// TIA Portal V17 export
// export: Created 2024-09-27T18:48:51.098157Z, ExportSetting WithDefaults, DisplayName Totally Integrated Automation Portal, DisplayVersion V17, DisplayName TIA Portal Openness, DisplayVersion V17, DisplayName TIA Portal Version Control Interface, DisplayVersion V17, DisplayName STEP 7 Professional, DisplayVersion V17, DisplayName STEP 7 Safety, DisplayVersion V17, DisplayName WinCC Professional, DisplayVersion V17
VAR_GLOBAL   // PLC tag table "Default tag table"
   i_PB_RESET_BEZPIECZENSTWA AT %I0.0 : Bool;
   i_KURTYNA_ŚWIETLNA_OK AT %I0.1 : Bool;
   i_E_STOP_OK AT %I0.2 : Bool;
   i_PB_START AT %I0.3 : Bool;
   i_PB_STOP AT %I0.4 : Bool;
   i_SIŁOWNIK_ZACISKAJĄCY_UGÓRY AT %I0.5 : Bool;
   i_SIŁOWNIK_ZACISKAJĄCY_W_DOLE AT %I0.6 : Bool;
   "i_SIŁOWNIK NASTAWY_GŁĘBOKIE" AT %I0.7 : Bool;
   "i_SIŁOWNIK NASTAWY _PŁYTKIE" AT %I1.0 : Bool;
   i_SIŁOWNIK_ODBIORU_POZ_STÓŁ AT %I1.1 : Bool;
   i_SIŁOWNIK_ODBIORU_POZ_ZRZUT AT %I1.2 : Bool;
   i_CZUJNIK_POZYCJI_STOŁU AT %I1.3 : Bool;
   i_CZUJNIK_SZTUKI_OK AT %I1.4 : Bool;
   i_CZUJNIK_PŁYTKIE_PRZÓD AT %I1.5 : Bool;
   Axis_1_Drive_IN AT %I68.0 : "PD_TEL3_IN";
   q_GŁÓWNY_ZAWÓR_POWIETRZA_ON AT %Q0.0 : Bool;
   q_NIEBIESKA_LAMPKA_SAFETY AT %Q0.1 : Bool;
   q_SIŁOWNIK_ZACISKAJĄCY_DOL AT %Q0.2 : Bool;
   q_EJECTOR_VACUM AT %Q0.3 : Bool;
   q_SIŁOWNIK_ZMIANY_GŁĘBOKIE AT %Q0.4 : Bool;
   q_EJECTOR_BLOWOFF AT %Q0.5 : Bool;
   q_SIŁOWNIK_ODBIERAJĄCY_STÓŁ AT %Q0.6 : Bool;
   q_LED_LAMP AT %Q0.7 : Bool;
   q_REZERWA1 AT %Q1.0 : Bool;
   q_REZERWA2 AT %Q1.1 : Bool;
   q_CZERWONA_KOLUMNA_SYGNALIZACYJNA AT %Q8.0 : Bool;
   q_ZÓŁTA_KOLUMNA_SYGNALIZACYJNA AT %Q8.1 : Bool;
   q_ZIELONA_KOLUMNA_SYGNALIZACYJNA AT %Q8.2 : Bool;
   q_BUZZER_KOLUMNA_SYGNALIZACYJNA AT %Q8.3 : Bool;
   q_SAFETY_RELAY_RESET AT %Q8.4 : Bool;
   q_REZERWA4 AT %Q8.5 : Bool;
   q_REZERWA5 AT %Q8.6 : Bool;
   q_REZERWA6 AT %Q8.7 : Bool;
   Clock_Byte AT %MB0 : Byte;
   Clock_10Hz AT %M0.0 : Bool;
   Clock_5Hz AT %M0.1 : Bool;
   "Clock_2.5Hz" AT %M0.2 : Bool;
   Clock_2Hz AT %M0.3 : Bool;
   "Clock_1.25Hz" AT %M0.4 : Bool;
   Clock_1Hz AT %M0.5 : Bool;
   "Clock_0.625Hz" AT %M0.6 : Bool;
   "Clock_0.5Hz" AT %M0.7 : Bool;
   m_SAFETY_OK AT %M1.0 : Bool;
   m_AUTO_MODE AT %M1.1 : Bool;
   m_SERVO_READY AT %M1.2 : Bool;
   MAN_SIŁ_ZAG_GÓRA AT %M1.3 : Bool;
   MAN_SIŁ_ZAG_DÓŁ AT %M1.4 : Bool;
   MAN_SIŁ_NASTAWY_GŁĘBOKIE AT %M1.5 : Bool;
   MAN_SIŁ_NASTAWY_PŁYTKIE AT %M1.6 : Bool;
   MAN_SIŁ_ODBIOR_STÓŁ AT %M1.7 : Bool;
   MAN_SIŁ_ODBIOR_ZRZUT AT %M2.0 : Bool;
   MAN_JOG_STOL_FWD AT %M2.1 : Bool;
   MAN_JOG_STOL_BWD AT %M2.2 : Bool;
   MAN_POZYCJA_STÓŁ_FWD AT %M2.3 : Bool;
   MAN_POZYCJA_STÓŁ_BWD AT %M2.4 : Bool;
   MAN_EJECTOR_SSANIE AT %M2.5 : Bool;
   MAN_EJECTOR_PRZEDMUCH AT %M2.6 : Bool;
   TP_ZAPISZ_WARTOŚĆ_PRED AT %M2.7 : Bool;
   TP_ZAPISZ_WARTOŚĆ_CZASU_PRZEDMUCHU AT %M3.0 : Bool;
   TP_ZAPISZ_WARTOSC_CZASU_SSANIA AT %M3.1 : Bool;
   TP_AKT_PRED_STOŁU AT %MW4 : Int;
   TP_NOWA_PRED_STOŁU AT %MW6 : Int;
   TP_AKT_CZAS_PRZEDMUCHU AT %MD50 : DInt;
   TP_NOWY_CZAS_PRZEDMUCHU AT %MD54 : DInt;
   TP_AKT_CZAS_SSANIA AT %MD58 : DInt;
   TP_NOWY_CZAS_SSANIA AT %MD62 : DInt;
   TP_LICZNIK_CAŁKOWITY AT %MD16 : DInt;
   TP_LICZNIK_ZADANE AT %MD20 : DInt;
   TP_LICZNIK_WYKONANE AT %MD24 : DInt;
   TP_KASUJ_LICZNIK_ZADANE AT %M3.2 : Bool;
   TP_USTAW_LICZNIK_ZADANE AT %M3.3 : Bool;
   TP_KASUJ_LICZNIK_AKTUALNE AT %M3.4 : Bool;
   m_STOL_KAT_OBROTU AT %MW28 : Int;
   TP_LED_ZAŁĄCZ AT %M3.5 : Bool;
   m_SRV_STO_ON AT %M3.6 : Bool;
   TP_USTAW_CZAS_TAKTU AT %M3.7 : Bool;
   AUTO_NUMER_KROKU AT %MW30 : Int;
   AUTO_KROK_1_ZAŁADUNEK AT %M32.0 : Bool;
   AUTO_KROK_2_OBRÓT_USTAW_GŁĘBOKIE AT %M32.1 : Bool;
   AUTO_KROK_3_ROZŁADUNEK AT %M32.2 : Bool;
   AUTO_KROK_4_ZJAZD_GŁĘBOKIE AT %M32.3 : Bool;
   AUTO_KROK_5_OBRÓT_USTAW_PLYTKIE AT %M32.4 : Bool;
   "AUTO_KROK_6_ZJAZD GŁOWICY PŁYTKIE" AT %M32.5 : Bool;
   AUTO_SERVO_FWD AT %M34.0 : Bool;
   AUTO_SIŁOWNIK_ZACISKAJĄCY_DÓŁ AT %M34.1 : Bool;
   AUTO_SIŁOWNIK_ZACISKAJĄCY_GÓRA AT %M34.2 : Bool;
   AUTO_SIŁOWNIK_NASTAWY_GŁĘBOKIE AT %M34.3 : Bool;
   AUTO_SIŁOWNIK_NASTAWY_PŁYTKIE AT %M34.4 : Bool;
   AUTO_SIŁOWNIK_ODBIORU_STÓŁ AT %M34.5 : Bool;
   AUTO_SIŁOWNIK_ODBIORU_ZRZUT AT %M34.6 : Bool;
   AUTO_EJECTOR_SSANIE AT %M34.7 : Bool;
   AUTO_EJECTOR_PRZEDMUCH AT %M35.0 : Bool;
   AUTO_TAKT_OBRÓT AT %MW38 : Int;
   TP_TAKT_ZADANA AT %MW40 : Int;
   TEST_BIT AT %M100.2 : Bool;
   TP_LAMP_TEST AT %M43.1 : Bool;
   m_TRYB_RĘCZNY_MOŻLIWY AT %M42.0 : Bool;
   MAN_Q_SIŁ_ZAG_GÓRA AT %M42.1 : Bool;
   MAN_Q_SIŁ_ZAG_DÓŁ AT %M42.2 : Bool;
   MAN_Q_SIŁ_NAS_GŁĘBOKIE AT %M42.3 : Bool;
   MAN_Q_SIŁ_NAS_PLYTKIE AT %M42.4 : Bool;
   MAN_Q_SIŁ_ODB_ZRZUT AT %M42.6 : Bool;
   MAN_Q_EJECTOR_SSANIE AT %M42.7 : Bool;
   MAN_Q_SIŁ_ODB_STÓŁ AT %M42.5 : Bool;
   MAN_Q_EJECTOR_PRZEDMUCH AT %M43.0 : Bool;
   m_ALARM_ACTIVE AT %M43.2 : Bool;
   m_WARNING_ACTIVE AT %M43.3 : Bool;
   AUTO_KROK2_WARUNKI_OK AT %M43.4 : Bool;
   m_ZBOCZE_P_POZ_STOŁU AT %M43.5 : Bool;
   m_ZBOCZE_P_CZUJNIK_SZTUK AT %M43.6 : Bool;
   AUTO_KROK5_WARUNKI_OK AT %M43.7 : Bool;
   AUTO_KROK6_WARUNKI_OK AT %M44.0 : Bool;
   TP_SCREEN_NO AT %MW46 : Int;
   System_Byte AT %MB1000 : Byte;
   FirstScan AT %M1000.0 : Bool;
   DiagStatusUpdate AT %M1000.1 : Bool;
   AlwaysTRUE AT %M1000.2 : Bool;
   AlwaysFALSE AT %M1000.3 : Bool;
   AUTO_CZAS_PRZEDMUCHU_SEK AT %MD66 : DInt;
   AUTO_CZAS_SSANIA_SEK AT %MD68 : DInt;
   test_power_in_enbl AT %M200.0 : Bool;
   TP_BTN_SET_HOME_POS AT %M358.3 : Bool;
   "temp_to pos_fwd" AT %M358.4 : Bool;
   temp_czujnik_poz_stolu_puls AT %M358.5 : Bool;
   "temp_to pos_bwd" AT %M358.6 : Bool;
   m_table_is_home AT %M358.7 : Bool;
   test_1 AT %M359.0 : Bool;
   test_2 AT %M359.1 : Bool;
   test_3 AT %M359.2 : Bool;
   test_4 AT %M359.3 : Bool;
   test_5 AT %M359.4 : Bool;
   test_6 AT %M359.5 : Bool;
   test_7 AT %M359.6 : Bool;
   test_8 AT %M359.7 : Bool;
   test_9 AT %M360.0 : Bool;
   test_10 AT %M360.1 : Bool;
   test_11 AT %M360.2 : Bool;
   test_12 AT %M360.3 : Bool;
   test_13 AT %M360.4 : Bool;
   test_14 AT %M360.5 : Bool;
   test_15 AT %M360.6 : Bool;
   test_16 AT %M360.7 : Bool;
   Axis_1_Drive_OUT AT %Q68.0 : "PD_TEL3_OUT";
   m_no_collision_table AT %M361.0 : Bool;
   TP_USTAW_DELAY_SIŁ_ZAG AT %M361.1 : Bool;
   TP_USTAW_DELAY_SIŁ_ODB AT %M361.2 : Bool;
   m_auto_table_velocity AT %MD362 : Real;
   m_memo_cycle_start AT %M8.0 : Bool;
   m_cycle_auto_possible AT %M8.1 : Bool;
   m_zbocze_N_kurtyna AT %M8.2 : Bool;
   m_auto_table_start_pos AT %M8.3 : Bool;
   m_zbocze_P_pb_start AT %M8.4 : Bool;
   m_zbocze_P_licznik AT %M8.5 : Bool;
   m_zbocze_P_licznik2 AT %M8.6 : Bool;
   tp_table_home_ok AT %M8.7 : Bool;
   m_memo_czujnik_stol_takt AT %M9.0 : Bool;
   m_memo_turn_started AT %M9.1 : Bool;
   m_auto_tact_time_elapsed AT %M9.2 : Bool;
   m_zbocze_N_czuj_stoł AT %M9.3 : Bool;
   m_memo_time_tack_elapsed AT %M9.4 : Bool;
   "m_auto_to pos_fwd" AT %M9.5 : Bool;
   temp_calc_new_tact AT %MD10 : Real;
   tp_display_akt_tact_time AT %MD72 : Real;
   m_zbocze_N_ustaw_takt AT %M9.6 : Bool;
   m_ustaw_takt_puls AT %M9.7 : Bool;
   tp_display_akt_sucktion_time AT %MD76 : Real;
   m_zbocze_N_ustaw_czas_ssania AT %M14.0 : Bool;
   tp_display_akt_blow_time AT %MD80 : Real;
   tp_display_akt_delay_sił_zag AT %MD84 : Real;
   tp_display_akt_delay_sił_odb AT %MD88 : Real;
   "m_zbocze_N-_czas_przedmuchu" AT %M14.1 : Bool;
   m_zboczeN_ustaw_delay_zagn AT %M14.2 : Bool;
   m_zboczeN_ustaw_delay_odbioru AT %M14.3 : Bool;
   m_zbocze_P_ustaw_czas_przedm AT %M14.4 : Bool;
   m_zbocze_P_delay_sił_zagniatania AT %M14.5 : Bool;
   m_auto_siłownik_odb_stoł AT %M14.6 : Bool;
   m_delay_sił_odbioru_elapsed AT %M14.7 : Bool;
   m_auto_zezwolenie_ssanie AT %M15.0 : Bool;
   m_delay_ssanie_elapsed AT %M15.1 : Bool;
   m_auto_zezwolenie_przedmuch AT %M15.2 : Bool;
   m_delay_przedmuch_elapsed AT %M15.3 : Bool;
   m_manual_mode AT %M15.4 : Bool;
   m_zbocze_czujnik_stołP2 AT %M15.5 : Bool;
   Flaga_nr_gniazda AT %M15.6 : Bool;
   m_zboczeN_zakon_przedmuch AT %M15.7 : Bool;
   m_potw_zakonczenia_rozł AT %M32.6 : Bool;
   m_zboczP_nowy_cykl_siłownika AT %M32.7 : Bool;
   m_memo_zboczeP_poz_odb AT %M33.0 : Bool;
   m_zbocze1 AT %M33.1 : Bool;
   m_zbocze2 AT %M33.2 : Bool;
   m_zbocze3 AT %M33.3 : Bool;
   m_auto_cycle_glebokie_gniazdo AT %M33.4 : Bool;
   m_auto_zmien_na_glebokie AT %M33.5 : Bool;
   m_zbocze4 AT %M33.6 : Bool;
   m_cycle5 AT %M33.7 : Bool;
   m_auto_sił_zagniatania_dol AT %M35.1 : Bool;
   m_auto_delay_zag_elapsed AT %M35.2 : Bool;
   m_stol_memo AT %M35.3 : Bool;
   m_zbocze5 AT %M35.4 : Bool;
   m_memo_kurtynaP AT %M35.5 : Bool;
   m_kurtyna_podczas_obrotu AT %M35.6 : Bool;
   m_sztuka_OK AT %M35.7 : Bool;
   m_obrót_krok AT %M36.0 : Bool;
   m_czujnik_ok AT %M36.1 : Bool;
   m_wykonano_zadana_ilosc AT %M36.2 : Bool;
   "m_powiadomienie_o zakonczeniu" AT %M36.3 : Bool;
   m_add_qty_cmpl AT %M36.4 : Bool;
   m_zboczeN_sztuki_OK AT %M36.5 : Bool;
   m_dodano AT %M36.6 : Bool;
   test1 AT %M36.7 : Bool;
END_VAR
